DEVICE_TYPE FRAME_DEVICE (* Top level window *)
  (* Standard: 61499-1 *)
  (* Version 0.2, 2001-11-25, JHC, Rockwell Automation, Corrected BOUNDS comment. *)
  (* Version 0.1, 2000-01-25, JHC, Rockwell Automation, Removed "Speed" Attribute *)
  (* Version 0.0, 2000-01-25, JHC, Rockwell Automation, Testing "Speed" Attribute *)
  (* Compiler header: package fb.rt.hmi;  import java.awt.*; *)
  (* Compiler Java IBM VisualAge 3.0 *)
  VAR_INPUT
    BOUNDS : ARRAY [0..3] OF DINT; (* Initial[x,y,width,height] *)
    GRID : ARRAY [0..1] OF DINT; (* Grid layout[rows,cols] *)
  END_VAR
END_DEVICE_TYPE
